// TIA Portal V16 export
// export: Created 2022-03-28T07:44:08.7630312Z, ExportSetting WithDefaults, DisplayName Totally Integrated Automation Portal, DisplayVersion V16 Update 5, DisplayName TIA Portal Version Control Interface, DisplayVersion V16 Update 2, DisplayName TIA Portal Openness, DisplayVersion V16 Update 5, DisplayName STEP 7 Professional, DisplayVersion V16 Update 5, DisplayName STEP 7 Safety, DisplayVersion V16, DisplayName WinCC Professional, DisplayVersion V16 Update 5
VAR_GLOBAL   // PLC tag table "Salidas PLC"
   Rearme AT %Q0.0 : Bool;
   "Marcha Soldadura" AT %Q0.1 : Bool;
   "Programa 1" AT %Q0.2 : Bool;
   "Programa 2" AT %Q0.3 : Bool;
   "Programa 4" AT %Q0.4 : Bool;
   "Programa 8" AT %Q0.5 : Bool;
   "Programa 16" AT %Q0.6 : Bool;
   "Reset error" AT %Q0.7 : Bool;
   Fluorescent AT %Q1.0 : Bool;
   "Piloto 1 Rojo" AT %Q2.0 : Bool;
   "Piloto 1 Ambar" AT %Q2.1 : Bool;
   "Piloto 1 Verde" AT %Q2.2 : Bool;
   "Piloto 2 Rojo" AT %Q2.3 : Bool;
   "Piloto 2 Ambar" AT %Q2.4 : Bool;
   "Piloto 2 Verde" AT %Q2.5 : Bool;
   "Piloto 3 Rojo" AT %Q2.6 : Bool;
   "Piloto 3 Ambar" AT %Q2.7 : Bool;
   "Piloto 3 Verde" AT %Q3.0 : Bool;
   "Baliza Roja" AT %Q3.1 : Bool;
   "Baliza Ambar" AT %Q3.2 : Bool;
   "Baliza Verde" AT %Q3.3 : Bool;
   "Pinza 1" AT %Q4.0 : Bool;
   "Pinza 2" AT %Q4.1 : Bool;
   "Pinza 3" AT %Q4.2 : Bool;
   "Piloto Marcha 1" AT %Q3.5 : Bool;
   "Piloto Marcha 2" AT %Q3.6 : Bool;
   "Piloto Marcha 3" AT %Q3.7 : Bool;
   "Piloto rearme" AT %Q3.4 : Bool;
   "Libre Q 4.7" AT %Q4.7 : Bool;
   Tag_46 AT %Q1.1 : Bool;
   bNotReady AT %Q4.4 : Bool;
   bRobotReset AT %Q4.5 : Bool;
END_VAR
